// TIA Portal V17 export
// export: Created 2023-04-04T13:27:32.688654Z, ExportSetting WithDefaults, DisplayName Totally Integrated Automation Portal, DisplayVersion V17, DisplayName TIA Portal Openness, DisplayVersion V17, DisplayName TIA Portal Version Control Interface, DisplayVersion V17, DisplayName STEP 7 Professional, DisplayVersion V17, DisplayName STEP 7 Safety, DisplayVersion V17, DisplayName WinCC Advanced, DisplayVersion V17
TYPE "typ_MQTT_Interface_Dashboard_Subscribe"
// stored: IsFailsafeCompliant false
   STRUCT
      Test : Bool;
      EnvironmentSensor : "typ_Environment_Sensor";
      BrightnessSensor { S7_SetPoint := 'True'} : "typ_Brightness_Sensor";
      CameraPicture { S7_SetPoint := 'True'} : "typ_Camera_Picture";
      PosPanTiltUnit { S7_SetPoint := 'True'} : "typ_Pos_Pan_Tilt_Unit_Enc";
      AlertMessage { S7_SetPoint := 'True'} : "typ_Alert_Message";
      Broadcast { S7_SetPoint := 'True'} : "typ_Broadcast";
      State_HBW : "typ_State_Client";
      State_VGR : "typ_State_Client";
      State_MPO : "typ_State_Client";
      State_SLD : "typ_State_Client";
      State_DSI : "typ_State_Client";
      State_DSO : "typ_State_Client";
      Stock_HBW { S7_SetPoint := 'True'} : "typ_Stock_Item";
      State_Order { S7_SetPoint := 'True'} : "typ_Order_Workpiece_Buttons_State";
      State_NFC_Device { S7_SetPoint := 'True'} : "typ_NFC_Module_State";
   END_STRUCT;
END_TYPE
